// This function has been automatically generated from the project information.
{attribute 'signature_flag' := '1073741824'}
{attribute 'TcGenerated'}
{attribute 'no-analysis'}
FUNCTION F_GetCompany : WSTRING
VAR_INPUT
	
END_VAR

F_GetCompany := "Beckhoff Automation LLC.";

END_FUNCTION

(* stored: Version 1.1.0.1
   POU F_GetCompany: Id {6ed15a98-db8c-4134-8548-07a6a0bdec12}, SpecialFunc None *)
